// TIA Portal V19 export
VAR_GLOBAL   // PLC tag table "3_BTRK_A0303_TRASFERIMENTO_LAYER_CONST"
END_VAR
VAR_GLOBAL CONSTANT   // user constants
   BTRK_A0303_TRASF_ATTESA_APERTO : Int := 1;
   BTRK_A0303_TRASF_ATTESA_CHIUSO : Int := 2;
END_VAR
